FUNCTION_BLOCK FB_HMI_TILT_B EXTENDS FB_HMI_COMPONENT
VAR_OUTPUT
END_VAR
VAR_IN_OUT
    fbInstance : FB_NOTT_TIP_TILT;
END_VAR
VAR
END_VAR

fbHealthStatus(

    bIsGood := NOT fbInstance.stat.bError,
    bHasWarning := (    fbInstance.stat.bWarning));
                     
fbBusyStatus(

    bIsBusy := FALSE);

M_UpdateStatusColor();

END_FUNCTION_BLOCK

(* stored: Version 1.1.0.1, ProductVersion 3.1.4024.14
   POU FB_HMI_TILT_B: Id {fb24523d-781d-4789-a662-3a43467d247d}, SpecialFunc None *)
